(* IEC 61131-3 sources: SRCI/RobotLibrary/RobotLibrary/POUs/Read/MC_ReadLoadData, 1 file *)

(* ---- MC_ReadLoadDataFB.st ---- *)
/// Read content of selected payload number
FUNCTION_BLOCK MC_ReadLoadDataFB EXTENDS RobotLibraryBaseExecuteFB
// -------------------------------------------------------------------------
//  SRCI Robot Library
// -------------------------------------------------------------------------
//
//  Object:      ReadLoadDataFB
//  Author:      Thorsten Brach
//  Date:        2024-06-01
//
//  Description:
//
//
//  Copyright:
//    (C) 2024 Thorsten Brach. All rights reserved
//             Licensed under the LGPL-3.0 license.
//
//  Disclaimer:
//    This project is provided without any guarantee and can be used for
//    private and commercial purposes. Any use is at the user’s
//    own risk and responsibility.
//
// -------------------------------------------------------------------------
VAR_INPUT
  /// command parameter
  ParCmd          : ReadLoadDataParCmd;
END_VAR
VAR_OUTPUT
  /// Command is transferred and confirmed by the RC
  CommandBuffered : BOOL;
  /// command outputs
  OutCmd          : ReadLoadDataOutCmd;
END_VAR

VAR
  /// internal copy of command parameter
 _parCmd          : ReadLoadDataParCmd;
  /// command data to send
 _command         : ReadLoadDataSendData;
  /// response data received
 _response        : ReadLoadDataRecvData;
END_VAR

  SUPER^(AxesGroup := AxesGroup);

END_FUNCTION_BLOCK

METHOD CheckParameterChanged : BOOL
VAR_IN_OUT
  /// Robot assignment of function
  AxesGroup    : AxesGroup;
END_VAR

  // Check ParCmd Size is > 0, becaue MemCmp does not work correctly with size = 0
  IF (SIZEOF(ParCmd) = 0)
  THEN
    RETURN;
  END_IF

  // compare memory
  CheckParameterChanged := ( MemCmp(ADR(ParCmd), ADR(_parCmd), SIZEOF(ParCmd)) <> RobotLibraryConstants.OK );

  IF ( CheckParameterChanged )
  THEN
    // update internal copy of parameters
   _parCmd := ParCmd;
    // inc parameter sequence
   _command.ParSeq := _command.ParSeq + 1;
    // update command data
    CommandData := CreateCommandPayload(); // ( Access via reference to rCommandFB in ACR )
    // notify active command register
    AxesGroup.Acyclic.ActiveCommandRegister.NotifyParameterChanged := _uniqueID;
  END_IF

END_METHOD

METHOD INTERNAL CreateCommandPayload : SendData
// Table 6-171: Sent CMD payload (PLC to RC) of "ReadLoadData"
// --------------------------
// Header
// --------------------------
// Byte 00 : UINT  - Type HB
// Byte 01 :       - Type LB
// Byte 02 : USINT - Reserve | ExecutionMode
// Byte 03 : USINT - ParSeq  | Priority
// --------------------------
// Datablock
// --------------------------
// Byte 04 : USINT  LoadNo;
// --------------------------

  // set command parameter
  _command.CmdTyp   :=  CmdType.ReadLoadData;
  _command.ExecMode :=  ExecMode;
  _command.ParSeq   := _command.ParSeq;
  _command.Priority :=  Priority;
  _command.LoadNo   := _parCmd.LoadNo;

  // copy command data to header
  _cmdHeader := _command;
  // call base implementation to copy header to payload buffer
  CreateCommandPayload := SUPER^.CreateCommandPayload();

  // add command.LoadNo
  CreateCommandPayload.AddInt(_command.LoadNo);

END_METHOD

METHOD FB_init : BOOL
VAR_INPUT
  /// if TRUE, the retain variables are initialized (warm start / cold start)
	bInitRetains : BOOL;
  /// if TRUE, the instance afterwards gets moved into the copy code (online change)
	bInCopyCode  : BOOL;
END_VAR

  MyType := 'MC_ReadLoadDataFB';

  ExecMode := ExecutionMode.PARALLEL;

END_METHOD

METHOD PROTECTED OnCall
VAR_IN_OUT
  /// Robot assignment of function
  AxesGroup : AxesGroup;
END_VAR

  // call base implementation
  SUPER^.OnCall(AxesGroup := AxesGroup);

  CASE _stepCmd OF

    00:  IF ( _execute_R.Q )
         THEN
           // set busy flag
           Busy := TRUE;
           // Reset command outputs
           MemSet(ADR(OutCmd),0,SIZEOF(OutCmd));
           // apply command parameter
          _parCmd := ParCmd;
           // init parameter sequence
          _command.ParSeq := 1;
           // set timeout
           SetTimeout(PT := _timeoutCmd, rTimer := _timerCmd);
           // inc step counter
          _stepCmd := _stepCmd + 1;
  	     END_IF

    01:  // create command data
         CommandData := CreateCommandPayload();
         // Add command to active command register
        _uniqueID := AxesGroup.Acyclic.ActiveCommandRegister.AddCmd( pCommandFB := ADR(THIS^ ));
         // set timeout
         SetTimeout(PT := _timeoutCmd, rTimer := _timerCmd);
         // inc step counter
        _stepCmd := _stepCmd + 1;

    02:  // Wait for responce received
         IF ( _responseReceived )
         THEN
           // reset response received flag
          _responseReceived := FALSE;

           CASE  _response.State
           OF
             CmdMessageState.BUFFERED : CommandBuffered := TRUE;
             CmdMessageState.DONE     : Done            := TRUE;
             CmdMessageState.ERROR    : Error           := TRUE;
  				 END_CASE

           // Done, Aborted or Error ?
           IF (_response.State >= CmdMessageState.DONE )
           THEN
             // Reset Busy flag
             Busy := FALSE;
             // Update results
             OutCmd.LoadNoReturn := _response.LoadNoReturn;
             OutCmd.LoadData     := _response.LoadData;
             // set timeout
             SetTimeout(PT := _timeoutCmd, rTimer := _timerCmd);
             // inc step counter
            _stepCmd := _stepCmd + 1;
  				 END_IF
         END_IF

    03: IF ( NOT Execute)
        THEN
          Reset();
  			END_IF
  ELSE
    // invalid step
    ErrorID := RobotLibraryEvents.ERR_INVALID_STEP;
  END_CASE

  // Cancel
  IF (Busy) AND (NOT Execute)
  THEN
    // try to remove cmd
    AxesGroup.Acyclic.ActiveCommandRegister.RemoveCmd(_uniqueID);
  END_IF

  // Reset FB
  IF ( NOT Execute )
  THEN
    Reset();
  END_IF

END_METHOD

METHOD INTERNAL ParseResponsePayload : DINT
// TTable 6-172: Received CMD payload (RC to PLC) of "ReadLoadData"
// --------------------------
// Header
// --------------------------
// Byte 00 : USINT   - ParSeq | State
// Byte 01 : SINT    - AlarmMessageSeverity
// Byte 02 : UINT    - AlarmMessageCode HB
// Byte 03 :         - AlarmMessageCode LB
// --------------------------
// Datablock
// --------------------------
// Byte 04 : DATE    - LoadData.Date LW HB;
// Byte 05 :         - LoadData.Date LW LB;
// Byte 06 : TOD     - LoadData.Time LW HB;
// Byte 07 :         - LoadData.Time LW LB;
// Byte 08 :         - LoadData.Time LW HB;
// Byte 09 :         - LoadData.Time LW LB;
// Byte 10 : REAL    - LoadData.X HW HB;
// Byte 11 :         - LoadData.X HW LB;
// Byte 12 :         - LoadData.X LW HB;
// Byte 13 :         - LoadData.X LW LB;
// Byte 14 : REAL    - LoadData.Y HW HB;
// Byte 15 :         - LoadData.Y HW LB;
// Byte 16 :         - LoadData.Y LW HB;
// Byte 17 :         - LoadData.Y LW LB;
// Byte 18 : REAL    - LoadData.Z HW HB;
// Byte 19 :         - LoadData.Z HW LB;
// Byte 20 :         - LoadData.Z LW HB;
// Byte 21 :         - LoadData.Z LW LB;
// Byte 22 : REAL    - LoadData.RX HW HB;
// Byte 23 :         - LoadData.RX HW LB;
// Byte 24 :         - LoadData.RX LW HB;
// Byte 25 :         - LoadData.RX LW LB;
// Byte 26 : REAL    - LoadData.RY HW HB;
// Byte 27 :         - LoadData.RY HW LB;
// Byte 28 :         - LoadData.RY LW HB;
// Byte 29 :         - LoadData.RY LW LB;
// Byte 30 : REAL    - LoadData.RZ HW HB;
// Byte 31 :         - LoadData.RZ HW LB;
// Byte 32 :         - LoadData.RZ LW HB;
// Byte 33 :         - LoadData.RZ LW LB;
// Byte 34 : REAL    - LoadData.Mass HW HB;
// Byte 35 :         - LoadData.Mass HW LB;
// Byte 36 :         - LoadData.Mass LW HB;
// Byte 37 :         - LoadData.Mass LW LB;
// Byte 38 : REAL    - LoadData.IX HW HB;
// Byte 39 :         - LoadData.IX HW LB;
// Byte 40 :         - LoadData.IX LW HB;
// Byte 41 :         - LoadData.IX LW LB;
// Byte 42 : REAL    - LoadData.IY HW HB;
// Byte 43 :         - LoadData.IY HW LB;
// Byte 44 :         - LoadData.IY LW HB;
// Byte 45 :         - LoadData.IY LW LB;
// Byte 46 : REAL    - LoadData.IZ HW HB;
// Byte 47 :         - LoadData.IZ HW LB;
// Byte 48 :         - LoadData.IZ LW HB;
// Byte 49 :         - LoadData.IZ LW LB;
// Byte 50 : USINT   - LoadNo;
// Byte 51 : BOOL    - DataChanged;
// --------------------------
VAR_INPUT
  /// Response data
  ResponseData : RecvData;
END_VAR

  // call base implementation to parse the header from payload buffer
  ResponseData.PayloadPtr := SUPER^.ParseResponsePayload(ResponseData);

  // copy parsed header to response
  _response.ParSeq               := _rspHeader.ParSeq;
  _response.State                := _rspHeader.State;
  _response.AlarmMessageSeverity := _rspHeader.AlarmMessageSeverity;
  _response.AlarmMessageCode     := _rspHeader.AlarmMessageCode;

  // Get Response.LoadData.Timestamp.IEC_DATE
  _response.LoadData.Timestamp.IEC_DATE := ResponseData.GetIecDate();
  // Get Response.LoadData.Timestamp.IEC_TIME
  _response.LoadData.Timestamp.IEC_TIME := ResponseData.GetIecTime();
  // Get Response.LoadData.X
  _response.LoadData.X := ResponseData.GetReal();
  // Get Response.LoadData.Y
  _response.LoadData.Y := ResponseData.GetReal();
  // Get Response.LoadData.Z
  _response.LoadData.Z := ResponseData.GetReal();
  // Get Response.LoadData.Rx
  _response.LoadData.Rx := ResponseData.GetReal();
  // Get Response.LoadData.Ry
  _response.LoadData.Ry := ResponseData.GetReal();
  // Get Response.LoadData.Rz
  _response.LoadData.Rz := ResponseData.GetReal();
  // Get Response.LoadData.Mass
  _response.LoadData.Mass := ResponseData.GetReal();
  // Get Response.LoadData.Ix
  _response.LoadData.Ix := ResponseData.GetReal();
  // Get Response.LoadData.Iy
  _response.LoadData.Iy := ResponseData.GetReal();
  // Get Response.LoadData.Iz
  _response.LoadData.Iz := ResponseData.GetReal();
  // Get Response.LoadNoReturn
  _response.LoadNoReturn := ResponseData.GetUsint();
  // Get Response.DataChanged
  _response.DataChanged := ResponseData.GetBool();

END_METHOD

METHOD PROTECTED Reset : DINT
VAR_INPUT
END_VAR

  Reset := SUPER^.Reset();

  Done               := FALSE;
  Busy               := FALSE;
  CommandBuffered    := FALSE;

END_METHOD
